(*Odd or none parity bit only in model  PMDLx-x-0/0.1.1.x.x*)
FUNCTION_BLOCK FB_TemperatureRelativeHumiditySensor_Emko EXTENDS FB_ModbusSlave

VAR
	lrTemperature	: LREAL;
	lrRelativeHumidity : LREAL;
END_VAR

METHOD Convert : BOOL
VAR_INPUT
	iRegionNo	:	INT;
	pReadData	:	POINTER TO word;
END_VAR
CASE iRegionNo OF
	0:
		lrTemperature := WORD_TO_LREAL( pReadData[0])*0.01;
		lrRelativeHumidity := WORD_TO_LREAL( pReadData[1])*0.1;
END_CASE
END_METHOD

METHOD FirstCycle // must be call once time 
VAR_INPUT
	sName : STRING;
	iUnitID : BYTE ; // modbus address of the device : 1- 255
END_VAR
SUPER^.FirstCycle( sName := sName,
					iUnitID := iUnitID);
arrAddress[0][0] := 0;
arrAddress[0][1] := 2;
arrAddress[0][2] := 1;
iNumAddRegion := 1;
iNumAddRegionWrite := 0;
END_METHOD

PROPERTY RelativeHumidity : lreal
GET
RelativeHumidity := lrRelativeHumidity;
END_GET
END_PROPERTY

PROPERTY Temperature : lreal
GET
Temperature := lrTemperature;
END_GET
END_PROPERTY

END_FUNCTION_BLOCK

(* stored: Version 1.1.0.1, ProductVersion 3.1.4024.12
   POU FB_TemperatureRelativeHumiditySensor_Emko: Id {0bf38bf5-d33e-4f48-84e4-db484ef3ee1d}, SpecialFunc None
   Method Convert: Id {5bb61268-8c5d-4e98-9923-f66dc8bd405e}
   Method FirstCycle: Id {b26eadeb-2397-4be7-a699-95ae1ee4a79f}
   Property RelativeHumidity: Id {27786f2a-dfae-44b2-9371-161830ee7879}
   Get Get: Id {b154d3f7-5429-4a10-8481-38209ff9d282}
   Property Temperature: Id {2f49b4d9-c379-4b1a-a23f-be051e0e6698}
   Get Get: Id {91c43331-e17f-4d5f-8db9-3e0490b10761} *)
